// TwinCAT 3 PLC project TcoRexrothPress
// Title: TcoRexrothPress
// Company: Vortex.Library
// ProjectVersion: 0.6.0.913
// ProgramVersion: 3.1.4023.0
// libraries:
//   Tc2_Standard, * (Beckhoff Automation GmbH)
//   Tc2_System, * (Beckhoff Automation GmbH)
//   Tc2_Utilities, * (Beckhoff Automation GmbH)
//   Tc3_Module, * (Beckhoff Automation GmbH)
//   TcoAbstractions, 0.6.0.913 (Vortex.Library)
//   TcoCore, 0.6.0.913 (Vortex.Library)
//   TcoIo, 0.6.0.913 (Vortex.Library)
//   TcoUtilities, 0.6.0.913 (Vortex.Library)
// project tree:
//   / PlcTask.TcTTO
//   POUs/SmartFunctionKit/IO/ TcoSmartFunctionKitIO_v_4_x_x.TcDUT, TcoSmartFunctionKitRequestHw_v_4_x_x.TcDUT, TcoSmartFunctionKitResponseHw_v_4_x_x.TcDUT
//   POUs/SmartFunctionKit/Structs/ eTcoSmartFunctionKitCommand_v_4_x_x.TcDUT, eTcoSmartFunctionKitParticipant_v_4_x_x.TcDUT, eTcoSmartFunctionKitStatusInformation_v_4_x_x.TcDUT, TcoSmartFunctionKitConfig_v_4_x_x.TcDUT, TcoSmartFunctionKitRequest_v_4_x_x.TcDUT, TcoSmartFunctionKitResponse_v_4_x_x.TcDUT, TcoSmartFunctionKitResults_v_4_x_x.TcDUT, TcoSmartFunctionKitStatus_v_4_x_x.TcDUT
//   POUs/SmartFunctionKit/Tasks/ TcoSmartFunctionKitCommand_v_4_x_x.TcPOU
//   POUs/SmartFunctionKit/ TcoSmartFunctionKit_v_4_x_x.TcPOU
// real-time tasks:
//   TASK PlcTask: cycle T#10ms, priority 20, ADS port 350
//   TASK PNIO: cycle T#16ms, priority 21, ADS port 351
//   TASK PlcTask1: cycle T#10ms, priority 22, ADS port 352
// I/O:
//   DEVICE Device 1 (EtherCAT) (disabled), AmsNetId 39.254.143.177.2.1
//     Press (IndraDrive MPC20 (1 CCD Master +0 CCD Slaves)) [IndraDrive MPC20 (1 CCD Master +0 CCD Slaves)]
// variable links:
//   TcoRexrothPressTests/TcoRexrothPressTests Instance <-> Device 1 (EtherCAT)/Press (IndraDrive MPC20 (1 CCD Master +0 CCD Slaves))
//     PlcTask Inputs/GVL_iXlinker.AdsAddr/netId <-> InfoData/AdsAddr/netId
//     PlcTask Inputs/GVL_iXlinker.AdsAddr/port <-> InfoData/AdsAddr/port
//     PlcTask Inputs/GVL_iXlinker.RexrothPress.Response.DigitalIoMapping <-> AT (CCD Master)/PLC output WORD8 AT %QB16
//     PlcTask Inputs/GVL_iXlinker.RexrothPress.Response.Handle <-> AT (CCD Master)/PLC output WORD4 AT %QB8
//     PlcTask Inputs/GVL_iXlinker.RexrothPress.Response.NotificationForce <-> AT (CCD Master)/PLC Global Register A24
//     PlcTask Inputs/GVL_iXlinker.RexrothPress.Response.NotificationId <-> AT (CCD Master)/PLC output WORD6 AT %QB12
//     PlcTask Inputs/GVL_iXlinker.RexrothPress.Response.NotificationPosition <-> AT (CCD Master)/Position feedback value 1
//     PlcTask Inputs/GVL_iXlinker.RexrothPress.Response.NotificationStatus <-> AT (CCD Master)/PLC output WORD7 AT %QB14
//     PlcTask Inputs/GVL_iXlinker.RexrothPress.Response.NotificationValue <-> AT (CCD Master)/PLC Global Register A23
//     PlcTask Inputs/GVL_iXlinker.RexrothPress.Response.NotificationVelocity <-> AT (CCD Master)/Velocity feedback value of encoder 1
//     PlcTask Inputs/GVL_iXlinker.RexrothPress.Response.Status <-> AT (CCD Master)/PLC output WORD5 AT %QB10
//     PlcTask Inputs/GVL_iXlinker.RexrothPress.Response.Value1 <-> AT (CCD Master)/PLC Global Register A20
//     PlcTask Inputs/GVL_iXlinker.RexrothPress.Response.Value2 <-> AT (CCD Master)/PLC Global Register A22
//     PlcTask Inputs/GVL_iXlinker.RexrothPress.Response.Value3 <-> AT (CCD Master)/PLC Global Register A21
//     PlcTask Inputs/GVL_iXlinker.RexrothPress.Response.VirtualIo <-> AT (CCD Master)/PLC output WORD9 AT %QB18
//     PlcTask Outputs/GVL_iXlinker.RexrothPress.Request.Command <-> MDT (CCD Master)/PLC input WORD5 AT %IB10
//     PlcTask Outputs/GVL_iXlinker.RexrothPress.Request.Handle <-> MDT (CCD Master)/PLC input WORD4 AT %IB8
//     PlcTask Outputs/GVL_iXlinker.RexrothPress.Request.Value1 <-> MDT (CCD Master)/PLC Global Register A17
//     PlcTask Outputs/GVL_iXlinker.RexrothPress.Request.Value2 <-> MDT (CCD Master)/PLC Global Register A18
//     PlcTask Outputs/GVL_iXlinker.RexrothPress.Request.Value3 <-> MDT (CCD Master)/PLC Global Register A19
//     PlcTask Outputs/GVL_iXlinker.RexrothPress.Request.Value7 <-> MDT (CCD Master)/PLC Global Register A25
//     PlcTask Outputs/GVL_iXlinker.RexrothPress.Request.Value4 <-> MDT (CCD Master)/PLC Global Register A4
//     PlcTask Outputs/GVL_iXlinker.RexrothPress.Request.Value5 <-> MDT (CCD Master)/PLC Global Register A5
//     PlcTask Outputs/GVL_iXlinker.RexrothPress.Request.Value6 <-> MDT (CCD Master)/PLC Global Register A6
//     PlcTask Outputs/GVL_iXlinker.RexrothPress.Request.VirtualIo <-> MDT (CCD Master)/PLC input WORD6 AT %IB12

CONFIGURATION TcoRexrothPress
    RESOURCE PLC ON TwinCAT3
        TASK PlcTask(INTERVAL := T#10ms, PRIORITY := 20);
        PROGRAM MAIN WITH PlcTask : MAIN;
    END_RESOURCE
END_CONFIGURATION

// ---- POUs/SmartFunctionKit/IO/TcoSmartFunctionKitIO_v_4_x_x.TcDUT
TYPE TcoSmartFunctionKitIO_v_4_x_x :
STRUCT
    Response : TcoSmartFunctionKitResponseHw_v_4_x_x;
    Request : TcoSmartFunctionKitRequestHw_v_4_x_x;
END_STRUCT
END_TYPE

// ---- POUs/SmartFunctionKit/IO/TcoSmartFunctionKitRequestHw_v_4_x_x.TcDUT
TYPE TcoSmartFunctionKitRequestHw_v_4_x_x :
STRUCT
    Handle AT %Q* : WORD;
    Command AT %Q* : WORD;
    Value1 AT %Q* : DWORD;
    Value2 AT %Q* : DWORD;
    Value3 AT %Q* : DWORD;
    Value4 AT %Q* : DWORD;
    Value5 AT %Q* : DWORD;
    Value6 AT %Q* : DWORD;
    Value7 AT %Q* : DWORD;
    VirtualIo AT %Q* : WORD;
END_STRUCT
END_TYPE

// ---- POUs/SmartFunctionKit/IO/TcoSmartFunctionKitResponseHw_v_4_x_x.TcDUT
TYPE TcoSmartFunctionKitResponseHw_v_4_x_x :
STRUCT
    Handle AT %I* : WORD;
    Status AT %I* : WORD;
    Value1 AT %I* : DWORD;
    Value2 AT %I* : DWORD;
    Value3 AT %I* : DWORD;
    NotificationId AT %I* : WORD;
    NotificationValue AT %I* : DWORD;
    NotificationStatus AT %I* : WORD;
    NotificationPosition AT %I* : DWORD;
    NotificationVelocity AT %I* : DWORD;
    NotificationForce AT %I* : DWORD;
    DigitalIoMapping AT %I* : WORD;
    VirtualIo AT %I* : WORD;
END_STRUCT
END_TYPE

// ---- POUs/SmartFunctionKit/Structs/eTcoSmartFunctionKitCommand_v_4_x_x.TcDUT
{attribute 'qualified_only'}
{attribute 'strict'}
TYPE eTcoSmartFunctionKitCommand_v_4_x_x :
(
    StartProgram := 1,
    SetProgramActive := 2,
    Positioning := 3,
    Jog := 4,
    ClearError := 5,
    StopMovement := 6,
    RestartDrive := 7,
    Tare := 9,
    StartHoming := 10,
    SetSystemVariable := 11,
    LockParticipant := 12,
    SetReference := 13,
    ReadSystemVariable := 14
);
END_TYPE

// ---- POUs/SmartFunctionKit/Structs/eTcoSmartFunctionKitParticipant_v_4_x_x.TcDUT
{attribute 'qualified_only'}
{attribute 'strict'}
TYPE eTcoSmartFunctionKitParticipant_v_4_x_x :
(
    WebInterface := 1,
    Fieldbus := 2,
    PhysicalInputsOutputs := 3
);
END_TYPE

// ---- POUs/SmartFunctionKit/Structs/eTcoSmartFunctionKitStatusInformation_v_4_x_x.TcDUT
{attribute 'qualified_only'}
{attribute 'strict'}
TYPE eTcoSmartFunctionKitStatusInformation_v_4_x_x :
(
    ActiveProgramNumber := 301, //  The PROGRAM number active in the drive is read out.
    RemainingStorageSpaceOnIPC := 302, // (PR21) The remaining storage space OF the IPC is transferred in MB.
    CurrentPosition := 401, //The cyclically transmitted position is read out.
    CurrentTravelSpeed := 402, // The cyclically transmitted travel speed is read out.
    CurrentForce := 403 // The cyclically transmitted force is read out
);
END_TYPE

// ---- POUs/SmartFunctionKit/Structs/TcoSmartFunctionKitConfig_v_4_x_x.TcDUT
TYPE TcoSmartFunctionKitConfig_v_4_x_x :
STRUCT
    DataFormat : eTcoDataFormat := TcoUtilities.eTcoDataFormat.BigEndian;
    InfoTime : TIME := T#2S;
    ErrorTime : TIME := T#5S;
    IpAddress : STRING;
    CurveExportLocation : STRING;
END_STRUCT
END_TYPE

// ---- POUs/SmartFunctionKit/Structs/TcoSmartFunctionKitRequest_v_4_x_x.TcDUT
TYPE TcoSmartFunctionKitRequest_v_4_x_x :
STRUCT
    Command : eTcoSmartFunctionKitCommand_v_4_x_x;
    SerialNumber : STRING(28);
    ProgramId : INT;
    PositionDistanceTara : REAL;
    TravelSpeed : REAL;
    Acceleration : REAL;
    Offset : REAL;
    Value1 : DWORD;
    Value2 : DWORD;
    Value3 : DWORD;
    Value4 : DWORD;
    Value5 : DWORD;
    Value6 : DWORD;
    Value7 : DWORD;
END_STRUCT
END_TYPE

// ---- POUs/SmartFunctionKit/Structs/TcoSmartFunctionKitResponse_v_4_x_x.TcDUT
TYPE TcoSmartFunctionKitResponse_v_4_x_x :
STRUCT
    AxisInReference : BOOL;
    ProgramActive : BOOL;
    LastPressingOk : BOOL;
    LastPressingNok : BOOL;
    SensorTared : BOOL;
    PressReady : BOOL;
    Error : BOOL;
    Warning : BOOL;
    RequestPossible : BOOL;
    ResponsAvialable : BOOL;
    NotificationAvailable : BOOL;
    EmergencyOffActive : BOOL;
    SafeStandstillActive : BOOL;
END_STRUCT
END_TYPE

// ---- POUs/SmartFunctionKit/Structs/TcoSmartFunctionKitResults_v_4_x_x.TcDUT
TYPE TcoSmartFunctionKitResults_v_4_x_x :
STRUCT
    id : STRING;
    maxForce : REAL;
    maxPosition : REAL;
    valid : BOOL;
    createdDate : DATE;
    cycleTime : REAL;
    validationTime : INT;
    status : STRING;
    customId : STRING;
    dataRecordingDisabled : BOOL;
    samplingInterval : INT;
    _v : INT;
END_STRUCT
END_TYPE

// ---- POUs/SmartFunctionKit/Structs/TcoSmartFunctionKitStatus_v_4_x_x.TcDUT
TYPE TcoSmartFunctionKitStatus_v_4_x_x :
STRUCT
    ActionDescription : STRING(100);
    ResponseStatus : TcoSmartFunctionKitResponse_v_4_x_x;
    NotificationId : UINT;
    NotificationToDisplay : eTcoSmartFunctionKitStatusInformation_v_4_x_x;
    NotificationPosition : REAL;
    NotificationVelocity : REAL;
    NotificationForce : REAL;
    DigitalIoMapping : DWORD;
    VirtualIo : DWORD;
END_STRUCT
END_TYPE

// ---- POUs/SmartFunctionKit/Tasks/TcoSmartFunctionKitCommand_v_4_x_x.TcPOU
FUNCTION_BLOCK TcoSmartFunctionKitCommand_v_4_x_x EXTENDS TcoCore.TcoTask
VAR_INPUT
    inCommand : TcoSmartFunctionKitRequest_v_4_x_x;
END_VAR
VAR_IN_OUT
    inoIoData : TcoSmartFunctionKitIO_v_4_x_x;
    inoConfig : TcoSmartFunctionKitConfig_v_4_x_x;
    inoStatus : TcoSmartFunctionKitStatus_v_4_x_x;
    inoResults : TcoSmartFunctionKitResults_v_4_x_x;
END_VAR
VAR
    {attribute 'hide'}
    _progress : INT := 0;
    {attribute 'hide'}
    _infoTimer : TON;
    {attribute 'hide'}
    _errorTimer : TON;
    {attribute 'hide'}
    _varInfo : __SYSTEM.VAR_INFO;
    {attribute 'hide'}
    _sb : TcoCore.StringBuilder;
END_VAR

IF Execute() THEN
    IF _progress = 0 THEN
        IF NOT __ISVALIDREF(inoIoData) THEN
            _varInfo := __VARINFO(inoIoData);
            Messenger.Programming(_sb.Clear().Append('<#Invalid reference: #>').Append(_varInfo.Symbol).ToString()).Pin();
        ELSIF NOT __ISVALIDREF(inoConfig) THEN
            _varInfo := __VARINFO(inoConfig);
            Messenger.Programming(_sb.Clear().Append('<#Invalid reference: #>').Append(_varInfo.Symbol).ToString()).Pin();
        ELSIF NOT __ISVALIDREF(inoStatus) THEN
            _varInfo := __VARINFO(inoStatus);
            Messenger.Programming(_sb.Clear().Append('<#Invalid reference: #>').Append(_varInfo.Symbol).ToString()).Pin();
        ELSIF NOT __ISVALIDREF(inoResults) THEN
            _varInfo := __VARINFO(inoResults);
            Messenger.Programming(_sb.Clear().Append('<#Invalid reference: #>').Append(_varInfo.Symbol).ToString()).Pin();
        ELSE
            _progress := _progress + 1;
        END_IF
    END_IF

    IF _progress = 1 THEN
        THIS^.inoStatus.ActionDescription := '<#Pressing running.#>';
        CallTimers(FALSE);
        THIS^.inoIoData.Request.Command := inCommand.Command;
        THIS^.inoIoData.Request.Value1 := inCommand.Value1;
        THIS^.inoIoData.Request.Value2 := inCommand.Value2;
        THIS^.inoIoData.Request.Value3 := inCommand.Value3;
        THIS^.inoIoData.Request.Value4 := inCommand.Value4;
        THIS^.inoIoData.Request.Value5 := inCommand.Value5;
        THIS^.inoIoData.Request.Value6 := inCommand.Value6;
        THIS^.inoIoData.Request.Value7 := inCommand.Value7;

        IF THIS^.inoStatus.ResponseStatus.RequestPossible THEN
            _progress := _progress + 1;
        END_IF;
    END_IF

    IF _progress = 2 THEN
        THIS^.inoIoData.Request.Handle := THIS^.inoIoData.Response.Handle + 1;

        IF THIS^.inoIoData.Request.Handle > 1000 THEN
            THIS^.inoIoData.Request.Handle := 1;
        END_IF

        _progress := _progress + 1;
    END_IF

    IF _progress = 3 THEN
        //THIS^.Messenger.OnCondition(_infoTimer.Q).Warning('<#Waiting for ProgramActive!#>').Pin();
        IF THIS^.inoIoData.Request.Handle <> THIS^.inoIoData.Response.Handle THEN
            _progress := _progress + 1;
        END_IF
    END_IF

    IF _progress = 4 THEN
        THIS^.Messenger.OnCondition(_infoTimer.Q AND THIS^.inoIoData.Response.Status = 0).Warning('<#Waiting for acknowledge Handle signal!#>');

        IF THIS^.inoIoData.Request.Handle = THIS^.inoIoData.Response.Handle AND THIS^.inoIoData.Response.Status = 0 THEN
            CallTimers(FALSE);
            _progress := 100;
        ELSIF THIS^.inoIoData.Request.Handle = THIS^.inoIoData.Response.Handle THEN
            IF THIS^.inoIoData.Response.Status <> 0 THEN
                Messenger.Build()
                    .Append('Function Smart Kit reported error: ')
                    .Append(TO_STRING(THIS^.inoIoData.Response.Status))
                    .Append(' |[[0]AdvancedDiagnosticMessage]|')
                    .As()
                    .AsError().Pin();
            END_IF

            THIS^.ThrowWhen(THIS^.inoIoData.Response.Status <> 0);
        END_IF
    END_IF

    IF _progress = 100 THEN
        THIS^.DoneWhen(TRUE);
        _progress := 0;
    END_IF

    CallTimers(TRUE);
    THIS^.ThrowWhen(_errorTimer.Q);
END_IF

METHOD CallTimers
VAR_INPUT
    inValue : BOOL;
END_VAR
IF __ISVALIDREF(inoConfig) THEN
    _infoTimer(IN := inValue, PT := THIS^.inoConfig.InfoTime);
    _errorTimer(IN := inValue, PT := THIS^.inoConfig.ErrorTime);
END_IF;
END_METHOD

{attribute 'hide'}
METHOD PUBLIC FB_init : BOOL
VAR_INPUT
    bInitRetains : BOOL; // if TRUE, the retain variables are initialized (warm start / cold start)
    bInCopyCode : BOOL; // if TRUE, the instance afterwards gets moved into the copy code (online change)
    ParentObject : ITcoObject;
END_VAR
END_METHOD

(*~
    <docu>
        <summary>
            Executes when task is aborted.
        </summary>
    </docu>
~*)
METHOD PROTECTED OnAbort
IF __ISVALIDREF(inoStatus) THEN
    THIS^.inoStatus.ActionDescription := '<#Pressing was aborted, while not yet completed!#>';
END_IF;
END_METHOD

(*~
    <docu>
        <summary>
            Executes when task reaches the ```Done``` state .
        </summary>
    </docu>
~*)
METHOD PROTECTED OnDone
IF __ISVALIDREF(inoStatus) THEN
    THIS^.inoStatus.ActionDescription := '<#Pressing was completed successfully.#>';
END_IF;
END_METHOD

(*~
    <docu>
        <summary>
            Executes when task reaches the ```Error``` state.
            <para>
                Do not confuse with <see cref="PlcDocu.TcoCore.TcoTask.WhileError()"/>, that is called cyclically until '''Error''' state is left.
            </para>
        </summary>
    </docu>
~*)
METHOD PROTECTED OnError
IF __ISVALIDREF(inoStatus) THEN
    THIS^.inoStatus.ActionDescription := '<#Pressing finished with error.#>';
END_IF;
END_METHOD

METHOD PROTECTED OnStart
IF __ISVALIDREF(inoStatus) THEN
    THIS^.inoStatus.ActionDescription := '<#Pressing started.#>';
END_IF;
END_METHOD

(*~
    <docu>
        <summary>
            Restores this instance to the Ready state. Can be called explicitly or from within one of the restore mechanisms.
            <para>
                See also <see cref="PlcDocu.TcoCore.TcoTask.AutoRestorable()"/>
            </para>
        </summary>
    </docu>
~*)
METHOD Restore : ITcoRestorable
SUPER^.Restore();
_progress := 0;
CallTimers(FALSE);
Messenger.UnPin();
END_METHOD

END_FUNCTION_BLOCK

// ---- POUs/SmartFunctionKit/TcoSmartFunctionKit_v_4_x_x.TcPOU
FUNCTION_BLOCK TcoSmartFunctionKit_v_4_x_x EXTENDS TcoIo.TcoEcatComponent
VAR_IN_OUT
    inoIoData : TcoSmartFunctionKitIO_v_4_x_x;
END_VAR
VAR
    {attribute addProperty Name "<#Config#>"}
    _config : TcoSmartFunctionKitConfig_v_4_x_x;
    {attribute addProperty Name "<#Status#>"}
    _status : TcoSmartFunctionKitStatus_v_4_x_x;
    _request : TcoSmartFunctionKitRequest_v_4_x_x;
    {attribute addProperty Name "<#Results#>"}
    _results : TcoSmartFunctionKitResults_v_4_x_x;
    converted : DWORD;
    i : INT;
    {attribute 'hide'}
    chars : ARRAY[0..MAX_STRING_LENGTH] OF BYTE;
    sCharacter : STRING(1) := '1';
END_VAR
VAR
    {attribute 'hide'}
    _taskEnabled : BOOL;
    {attribute addProperty Name "<#Run Command#>"}
    _runCommandTask : TcoSmartFunctionKitCommand_v_4_x_x(THIS^);
    {attribute addProperty Name "<#Get last Results#>" }
    _getResultsTask : TcoCore.TcoRemoteTask(THIS^);
    {attribute addProperty Name "<#Save last curve#>" }
    _exportCurveTask : TcoCore.TcoRemoteTask(THIS^);
    {attribute addProperty Name "<#Restore Task#>"}
    _restoreTask : TcoCore.TcoTask(THIS^);
END_VAR
VAR
    {attribute 'hide'}
    _varInfo : __SYSTEM.VAR_INFO;
    {attribute 'hide'}
    _amsId : STRING(23);
END_VAR

IF InvalidReference() THEN
    RETURN;
END_IF

SUPER^(AdsAddr := AdsAddr);
UpdateResponses();

CASE _request.Command OF
    eTcoSmartFunctionKitCommand_v_4_x_x.StartProgram:
        chars := MAXSTRING_TO_BYTEARR(_request.SerialNumber);

        FOR i := LEN(_request.SerialNumber) + 1 TO 255 BY 1 DO
            chars[i] := 0;
        END_FOR;

        i := 0;

        _request.Value1 := THIS^._BYTES_TO_DWORD(Format := _config.DataFormat,
            INb0 := chars[i],
            INb1 := chars[i + 1],
            INb2 := chars[i + 2],
            INb3 := chars[i + 3]);

        i := 4;

        _request.Value2 := THIS^._BYTES_TO_DWORD(Format := _config.DataFormat,
            INb0 := chars[i],
            INb1 := chars[i + 1],
            INb2 := chars[i + 2],
            INb3 := chars[i + 3]);

        i := 8;

        _request.Value3 := THIS^._BYTES_TO_DWORD(Format := _config.DataFormat,
            INb0 := chars[i],
            INb1 := chars[i + 1],
            INb2 := chars[i + 2],
            INb3 := chars[i + 3]);

        i := 12;

        _request.Value4 := THIS^._BYTES_TO_DWORD(Format := _config.DataFormat,
            INb0 := chars[i],
            INb1 := chars[i + 1],
            INb2 := chars[i + 2],
            INb3 := chars[i + 3]);

        i := 16;

        _request.Value5 := THIS^._BYTES_TO_DWORD(Format := _config.DataFormat,
            INb0 := chars[i],
            INb1 := chars[i + 1],
            INb2 := chars[i + 2],
            INb3 := chars[i + 3]);

        i := 20;

        _request.Value6 := THIS^._BYTES_TO_DWORD(Format := _config.DataFormat,
            INb0 := chars[i],
            INb1 := chars[i + 1],
            INb2 := chars[i + 2],
            INb3 := chars[i + 3]);

        i := 24;

        _request.Value7 := THIS^._BYTES_TO_DWORD(Format := _config.DataFormat,
            INb0 := chars[i],
            INb1 := chars[i + 1],
            INb2 := chars[i + 2],
            INb3 := chars[i + 3]);
    eTcoSmartFunctionKitCommand_v_4_x_x.SetProgramActive:
        _request.Value1 := INT_TO_DWORD(_request.ProgramId * 1000);
    eTcoSmartFunctionKitCommand_v_4_x_x.Positioning:
        _request.Value1 := REAL_TO_DWORD(_request.PositionDistanceTara * 1000);
        _request.Value2 := REAL_TO_DWORD(_request.TravelSpeed * 1000);
        _request.Value3 := REAL_TO_DWORD(_request.Acceleration * 1000);
    eTcoSmartFunctionKitCommand_v_4_x_x.Jog:
        _request.Value1 := REAL_TO_DWORD(_request.PositionDistanceTara * 1000);
        _request.Value2 := REAL_TO_DWORD(_request.TravelSpeed * 1000);
        _request.Value3 := REAL_TO_DWORD(_request.Acceleration * 1000);
    eTcoSmartFunctionKitCommand_v_4_x_x.Tare:
        _request.Value1 := REAL_TO_DWORD(_request.Offset * 1000);
END_CASE
//*************READ***********************
_taskEnabled := TRUE;
_taskEnabled := _taskEnabled;
_runCommandTask.Enabled := _taskEnabled;

_runCommandTask(inCommand := _request,
    inoIoData := THIS^.inoIoData,
    inoConfig := THIS^._config,
    inoStatus := THIS^._status,
    inoResults := THIS^._results);
//****************************************
//*************RESTORE********************
_taskEnabled := TRUE;
_restoreTask.Enabled := _taskEnabled;

IF _restoreTask.Execute() THEN
    Restore();
END_IF
//****************************************
_exportCurveTask();
_getResultsTask();

METHOD _BYTES_TO_DWORD : DWORD
VAR_INPUT
    Format : TcoUtilities.eTcoDataFormat;
    INb0 : BYTE;
    INb1 : BYTE;
    INb2 : BYTE;
    INb3 : BYTE;
END_VAR
VAR
    b0 : BYTE;
    b1 : BYTE;
    b2 : BYTE;
    b3 : BYTE;
    tmpDWORD : DWORD;
END_VAR
IF Format = TcoUtilities.eTcoDataFormat.LittleEndian THEN
    b0 := INb3;
    b1 := INb2;
    b2 := INb1;
    b3 := INb0;
ELSIF Format = TcoUtilities.eTcoDataFormat.BigEndian THEN
    b0 := INb0;
    b1 := INb1;
    b2 := INb2;
    b3 := INb3;
END_IF

tmpDWORD := b0;
tmpDWORD := SHL(tmpDWORD, 8);
tmpDWORD := tmpDWORD + b1;
tmpDWORD := SHL(tmpDWORD, 8);
tmpDWORD := tmpDWORD + b2;
tmpDWORD := SHL(tmpDWORD, 8);
tmpDWORD := tmpDWORD + b3;
_BYTES_TO_DWORD := tmpDWORD;
END_METHOD

(*~
    <docu>
        <summary>
            Gets the configuration of the SFK.
        </summary>
    </docu>
~*)
PROPERTY Config : REFERENCE TO TcoSmartFunctionKitConfig_v_4_x_x
GET
Config REF= _config;
END_GET
END_PROPERTY

(*~
    <docu>
        <summary>
            Run specified comand of smart function kit.
        </summary>
    </docu>
~*)
METHOD ExportLastCurve : TcoCore.ITcoTaskStatus
ExportLastCurve := THIS^._exportCurveTask.Invoke();
END_METHOD

(*~
    <docu>
        <summary>
            Gets the `ReadTask` task that controls the reading sequence.
        </summary>
    </docu>
~*)
PROPERTY ExportLastCurveTask : REFERENCE TO TcoCore.TcoRemoteTask
GET
ExportLastCurveTask ref= _exportCurveTask;
END_GET
END_PROPERTY

METHOD FB_init : BOOL
VAR_INPUT
    bInitRetains : BOOL; // if TRUE, the retain variables are initialized (warm start / cold start)
    bInCopyCode : BOOL; // if TRUE, the instance afterwards gets moved into the copy code (online change)
    ParentObject : ITcoObject;
END_VAR
END_METHOD

METHOD GetResults : TcoCore.ITcoTaskStatus
VAR_INPUT
END_VAR
GetResults := this^._getResultsTask.Invoke();
END_METHOD

(*~
    <docu>
        <summary>
            Gets the `ReadTask` task that controls the reading sequence.
        </summary>
    </docu>
~*)
PROPERTY GetResultsTask : REFERENCE TO TcoCore.TcoRemoteTask
GET
GetResultsTask ref= _getResultsTask;
END_GET
END_PROPERTY

METHOD INTERNAL InvalidReference : BOOL
InvalidReference := FALSE;

IF NOT __ISVALIDREF(inoIoData) THEN
    _varInfo := __VARINFO(inoIoData);
    Messenger.Error(_sb.Clear().Append('<#Invalid reference: #>').Append(_varInfo.Symbol).ToString());
    InvalidReference := TRUE;
END_IF
END_METHOD

(*~
    <docu>
        <summary>
            Gets the configuration of the SFK.
        </summary>
    </docu>
~*)
PROPERTY Request : REFERENCE TO TcoSmartFunctionKitRequest_v_4_x_x
GET
Request REF= _request;
END_GET
END_PROPERTY

(*~
    <docu>
        <summary>
            Restores this instance to the Ready state. Can be called explicitly or from within one of the restore mechanisms.
        </summary>
    </docu>
~*)
METHOD Restore : ITcoRestorable
IF InvalidReference() THEN
    RETURN;
END_IF

_restoreTask.Restore();
_ecatState.Restore();
_runCommandTask.Restore();
_getResultsTask.Restore();
_exportCurveTask.Restore();
Tc2_System.MEMSET(destAddr := ADR(THIS^.inoIoData), fillByte := 0, n := SIZEOF(THIS^.inoIoData));
_status.ActionDescription := '<#Restore executed!#>';
inoIoData.Request.Command := 0;
inoIoData.Request.VirtualIo := 0;
inoIoData.Request.Value1 := 0;
inoIoData.Request.Value2 := 0;
inoIoData.Request.Value3 := 0;
inoIoData.Request.Value4 := 0;
inoIoData.Request.Value5 := 0;
inoIoData.Request.Value6 := 0;
inoIoData.Request.Value7 := 0;
END_METHOD

(*~
    <docu>
        <summary>
            Run specified comand of smart function kit.
        </summary>
    </docu>
~*)
METHOD RunCommand : TcoCore.ITcoTaskStatus
RunCommand := THIS^._runCommandTask.Invoke();
END_METHOD

(*~
    <docu>
        <summary>
            Gets the `ReadTask` task that controls the reading sequence.
        </summary>
    </docu>
~*)
PROPERTY RunCommandTask : TcoCore.ITcoTaskStatus
GET
RunCommandTask := _runCommandTask;
END_GET
END_PROPERTY

(*~
    <docu>
        <summary>
            Custom service (manual, maintenance) logic.
            This method must be implemented in derived class.
        </summary>
    </docu>
~*)
METHOD PROTECTED ServiceMode
END_METHOD

(*~
    <docu>
        <summary>
            Gets the status of the SFK.
        </summary>
    </docu>
~*)
PROPERTY Status : REFERENCE TO TcoSmartFunctionKitStatus_v_4_x_x
GET
Status REF= _status;
END_GET
END_PROPERTY

METHOD INTERNAL UpdateResponses
VAR
    enumVal : eTcoSmartFunctionKitStatusInformation_v_4_x_x;
END_VAR
_status.ResponseStatus.AxisInReference := inoIoData.Response.NotificationStatus.2;
_status.ResponseStatus.ProgramActive := inoIoData.Response.NotificationStatus.3;
_status.ResponseStatus.LastPressingOk := inoIoData.Response.NotificationStatus.4;
_status.ResponseStatus.LastPressingNok := inoIoData.Response.NotificationStatus.5;
_status.ResponseStatus.SensorTared := inoIoData.Response.NotificationStatus.6;
_status.ResponseStatus.PressReady := inoIoData.Response.NotificationStatus.7;
_status.ResponseStatus.Error := inoIoData.Response.NotificationStatus.8;
_status.ResponseStatus.Warning := inoIoData.Response.NotificationStatus.9;
_status.ResponseStatus.RequestPossible := inoIoData.Response.NotificationStatus.11;
_status.ResponseStatus.ResponsAvialable := inoIoData.Response.NotificationStatus.12;
_status.ResponseStatus.NotificationAvailable := inoIoData.Response.NotificationStatus.13;
_status.ResponseStatus.EmergencyOffActive := inoIoData.Response.NotificationStatus.14;
_status.ResponseStatus.SafeStandstillActive := inoIoData.Response.NotificationStatus.15;
_status.NotificationPosition := DWORD_TO_REAL(inoIoData.Response.NotificationPosition) / 10000;
_status.NotificationVelocity := DWORD_TO_REAL(inoIoData.Response.NotificationVelocity) / 10000;
_status.NotificationForce := DWORD_TO_REAL(inoIoData.Response.NotificationForce) / 1000;
_status.NotificationId := inoIoData.Response.NotificationId;

CASE inoIoData.Response.NotificationId of
    eTcoSmartFunctionKitStatusInformation_v_4_x_x.ActiveProgramNumber:
        enumVal := eTcoSmartFunctionKitStatusInformation_v_4_x_x.ActiveProgramNumber;
    eTcoSmartFunctionKitStatusInformation_v_4_x_x.CurrentForce:
        enumVal := eTcoSmartFunctionKitStatusInformation_v_4_x_x.CurrentForce;
    eTcoSmartFunctionKitStatusInformation_v_4_x_x.CurrentPosition:
        enumVal := eTcoSmartFunctionKitStatusInformation_v_4_x_x.CurrentPosition;
    eTcoSmartFunctionKitStatusInformation_v_4_x_x.CurrentTravelSpeed:
        enumVal := eTcoSmartFunctionKitStatusInformation_v_4_x_x.CurrentTravelSpeed;
    eTcoSmartFunctionKitStatusInformation_v_4_x_x.RemainingStorageSpaceOnIPC:
        enumVal := eTcoSmartFunctionKitStatusInformation_v_4_x_x.RemainingStorageSpaceOnIPC;
END_CASE

_status.NotificationToDisplay := enumVal;
_status.DigitalIoMapping := inoIoData.Response.DigitalIoMapping;
END_METHOD

END_FUNCTION_BLOCK
